// TwinCAT 3 PLC project FileReader_Test
// ProgramVersion: 3.1.4026.12
// libraries:
//   SH_FileReader, * (Stefan Halder)
//   Tc2_Standard, * (Beckhoff Automation GmbH)
//   Tc2_System, * (Beckhoff Automation GmbH)
// project tree:
//   / PlcTask.TcTTO
//   POUs/ MAIN.TcPOU
// (motion and I/O tree: see PLC project sh_filereader)
// real-time tasks:
//   TASK PlcTask: cycle T#10ms, priority 20, ADS port 350

CONFIGURATION FileReader_Test
    RESOURCE PLC ON TwinCAT3
        TASK PlcTask(INTERVAL := T#10ms, PRIORITY := 20);
        PROGRAM MAIN WITH PlcTask : MAIN;
    END_RESOURCE
END_CONFIGURATION

// ---- POUs/MAIN.TcPOU
PROGRAM MAIN
VAR
	fb_FileReader : SH_FileReader.FileReader;
	
	bReadFile : BOOL;
	sFilePath : STRING := 'E:\Projects\Twincat\AdventOfCode\Day02\Day2Input.txt';
	bFileReaderDone : BOOL;
	stError : SH_FileReader.ERROR;
END_VAR

fb_FileReader();


bFileReaderDone := fb_FileReader.ReadFile(bExecute := bReadFile, sFilePath := sFilePath, stError => stError);
IF bReadFile THEN
	bReadFile := FALSE;
END_IF

END_PROGRAM
